SUBAPPLICATION Uebung_226_AX (* Split-Bargraph (wie Uebung_226 in test_B, aber mit AR-Adapter-Baustein BargraphSplitFS_AR statt REQ/rValue) *)
  (* Standard: 61499-2; Description: Copyright (c) 2026 Meisterschulen am Ostbahnhof This program and the accompanying materials are made available under the terms of the Eclipse Public License 2.0 which is available at https://www.eclipse.org/legal/epl-2.0/ SPDX-License-Identifier: EPL-2.0 *)
  (* Version 1.0, 2026-09-05, Franz Höpfinger, Meisterschulen am Ostbahnhof, adapter variant of Uebung_226 (test_B) using NumericValue_PHYSA/BargraphSplitFS_AR *)
  PACKAGE Uebungen;
  IMPORT Uebungen::const::UT::Dreieck::DefaultPool_Dreieck_BargraphSplit::Bargraph_Split_BargraphSplit;
  IMPORT Uebungen::const::UT::Dreieck::DefaultPool_Dreieck_Numeric::NumberVariable_Sollwert_N;
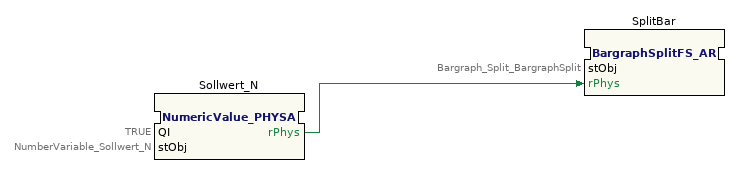
  FBS
    Sollwert_N : isobus::UT::io::NumericValue::NumericValue_PHYSA(QI := TRUE, stObj := NumberVariable_Sollwert_N);
    SplitBar : isobus::UT::Q::BargraphSplitFS_AR(stObj := Bargraph_Split_BargraphSplit);
  END_FBS
  ADAPTER_CONNECTIONS
    Sollwert_N.rPhys TO SplitBar.rPhys;
  END_CONNECTIONS
END_SUBAPPLICATION
